// Mitsubishi GX Works2 project: Helloworldtentativa1   PLC: Q03UDV

PROGRAM MAIN
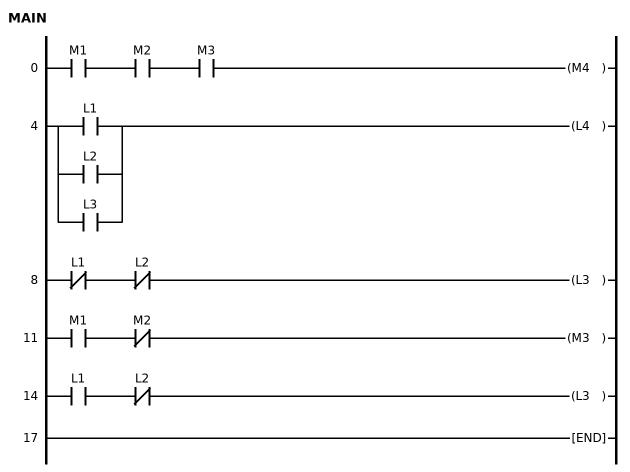
0     LD      M1
      AND     M2
      AND     M3
      OUT     M4
4     LD      L1
      OR      L2
      OR      L3
      OUT     L4
8     LDI     L1
      ANI     L2
      OUT     L3
11    LD      M1
      ANI     M2
      OUT     M3
14    LD      L1
      ANI     L2
      OUT     L3
17    END
END_PROGRAM
